// TIA Portal V18 export
// export: Created 2026-06-09T02:47:52.5688093Z, ExportSetting WithDefaults, DisplayName Totally Integrated Automation Portal, DisplayVersion V18, DisplayName TIA Portal Openness, DisplayVersion V18, DisplayName TIA Portal Version Control Interface, DisplayVersion V18, DisplayName STEP 7 Professional, DisplayVersion V18, DisplayName STEP 7 Safety, DisplayVersion V18, DisplayName WinCC Professional, DisplayVersion V18
VAR_GLOBAL   // PLC tag table "Etykieciarka"
   start_etykieciarka AT %M102.0 : Bool;
   stop_etykieciarka AT %M102.1 : Bool;
   cz_swiatlowodowy AT %M202.0 : Bool;
   etykieta AT %Q0.6 : Bool;
   tasma_etykieciarka AT %Q0.7 : Bool;
   lampa_sygnalizacyjna_etyk AT %Q1.0 : Bool;
END_VAR
